FUNCTION_BLOCK PAEActValve3 EXTENDS PAEActuator3way
VAR_INPUT
END_VAR
VAR_OUTPUT
END_VAR
VAR
END_VAR

METHOD PUBLIC PAEActValve3
VAR_INPUT
END_VAR
END_METHOD

END_FUNCTION_BLOCK

(* stored: Version 1.1.0.1, ProductVersion 3.1.4020.12
   POU PAEActValve3: Id {e6651301-b59d-4be3-8af8-554efbcae8cf}, SpecialFunc None
   Method PAEActValve3: Id {b9e13882-5884-4929-92f5-16b941aed5d8} *)
